// TIA Portal V17 export
// export: Created 2022-04-06T07:28:41.2047537Z, ExportSetting WithDefaults, DisplayName Totally Integrated Automation Portal, DisplayVersion V17, DisplayName TIA Portal Openness, DisplayVersion V17, DisplayName TIA Portal Version Control Interface, DisplayVersion V17, DisplayName TIA Portal Test Suite Advanced, DisplayVersion V17, DisplayName SINAMICS Startdrive Advanced, DisplayVersion V17, DisplayName SINAMICS Startdrive G130, G150, S120, S150, SINAMICS MV, S210, DisplayVersion V17, DisplayName SINAMICS Startdrive G110M, G120, G120C, G120D, G120P, G115D, DisplayVersion V17, DisplayName STEP 7 Professional, DisplayVersion V17, DisplayName STEP 7 Safety, DisplayVersion V17, DisplayName WinCC Advanced / Unified PC, DisplayVersion V17
TYPE "LAxisCtrl_typeGeneralSettings"
TITLE = LAxisCtrl_typeGeneralSettings
// Support: tech.team.motioncontrol@siemens.com
// stored: IsFailsafeCompliant false
   STRUCT
      stopOnError : Bool := TRUE;   // TRUE: In case of error the axis will be stopped automatically with fastStop dynamics
      resetWithRestart : Bool := FALSE;   // TRUE: Reinitialization of the technology object and acknowledgment of pending technology alarms. The technology object is reinitialized with the configured start values; FALSE: Acknowledgment of queued technology alarms
      abortWaitingSyncCmd : Bool := TRUE;   // TRUE: Abort waiting synchronous command in case of new basic motion command automatically
   END_STRUCT;
END_TYPE
